//==================================================================================================
//								RJM Maszyny sp. z o.o.
//									13.05.2022
//	Obsługa silonwika podstawa z kontrolą czasów oraz kontrolą czujników
//	Realizacja wysuwania i chowania tłoczyska dla jednej cewki zwrócenie pozycji skrajnych
// 	v1.0	|| TC v 3.1.4024.22		|| - pierwsza wersja
//==================================================================================================
FUNCTION_BLOCK FB_Silownik_Kontola EXTENDS FB_Silownik 
VAR_INPUT
	stParametry								: DUT_SilownikParametry;
END_VAR
VAR_OUTPUT
END_VAR
VAR
	tonCzasNaPrace							: TON;
	tonCzasNaPowrot							: TON;
	fbKontrolaCzujnik0_F					: F_TRIG;
	fbKontrolaCzujnikMax_F					: F_TRIG;
	fbKontrolaCzujnik0_R					: R_TRIG;
	fbKontrolaCzujnikMax_R					: R_TRIG;
	fbLBKomunikacja							: FB_Silownik_Kontrola_Komunikacja;
END_VAR

METHOD Praca : BOOL
VAR_INPUT
END_VAR
SUPER^.Praca ();
//Czasy sprawdzające czas wysunięcia lub chowania tłoczyska
	tonCzasNaPrace (IN := bPrzesuwanieWStroneKonca, PT := REAL_TO_TIME (stParametry.rCzasNaPrace));
	tonCzasNaPowrot (In := bPrzesuwanieWStronePoczatku, PT := REAL_TO_TIME (stParametry.rCzasNaPowrot));
//kontrola wysuwania
	IF (tonCzasNaPrace.Q) THEN
		fbLBKomunikacja.UstawStan (iId := 1, bStan := TRUE);
	ELSIF (fbCzujnikPozycjaMax.CzyZadzialany AND NOT bPrzesuwanieWStroneKonca) THEN
		fbLBKomunikacja.UstawStan (iId := 1, bStan := FALSE);
	END_IF
//kontrola powrotu
	IF (tonCzasNaPowrot.Q) THEN
		fbLBKomunikacja.UstawStan (iId := 2, bStan := TRUE);
	ELSIF (fbCzujnikPozycja0.CzyZadzialany AND NOT bPrzesuwanieWStronePoczatku) THEN
		fbLBKomunikacja.UstawStan (iId := 2, bStan := FALSE);
	END_IF
//kontrola utraty pozycji 0
	fbKontrolaCzujnik0_F (CLK := fbCzujnikPozycja0.CzyZadzialany);
	IF (fbKontrolaCzujnik0_F.Q AND NOT bPrzesuwanieWStroneKonca) THEN
		fbLBKomunikacja.UstawStan (iId := 3, bStan := TRUE);
	ELSIF (fbCzujnikPozycja0.CzyZadzialany) THEN
		fbLBKomunikacja.UstawStan (iId := 3, bStan := FALSE);
	END_IF
//kontrola utraty pozycji MAX
	fbKontrolaCzujnikMax_F (CLK := fbCzujnikPozycjaMax.CzyZadzialany);
	IF (fbKontrolaCzujnikMax_F.Q AND NOT bPrzesuwanieWStronePoczatku) THEN
		fbLBKomunikacja.UstawStan (iId := 4, bStan := TRUE);
	ELSIF (fbCzujnikPozycjaMax.CzyZadzialany) THEN
		fbLBKomunikacja.UstawStan (iId := 4, bStan := FALSE);
	END_IF	
//Bladustawienia czujnikow - zadziałane dwa czujniki
	IF (fbCzujnikPozycja0.CzyZadzialany AND fbCzujnikPozycjaMax.CzyZadzialany) THEN
		fbLBKomunikacja.UstawStan (iId := 5, bStan := TRUE);
	ELSE
		fbLBKomunikacja.UstawStan (iId := 5, bStan := FALSE);
	END_IF
//Blad zamiany czujnikow	
	fbKontrolaCzujnik0_R (CLK := fbCzujnikPozycja0.CzyZadzialany);
	fbKontrolaCzujnikMax_R (CLK := fbCzujnikPozycjaMax.CzyZadzialany);
	IF ((fbKontrolaCzujnik0_R.Q AND bPrzesuwanieWStroneKonca) OR
		(fbKontrolaCzujnikMax_R.Q AND bPrzesuwanieWStronePoczatku)) THEN
		fbLBKomunikacja.UstawStan (iId := 6, bStan := FALSE);
	END_IF
	IF ((NaPoczatku AND NOT bPrzesuwanieWStroneKonca) OR 
		(NaKoncu and not bPrzesuwanieWStronePoczatku) ) THEN
		fbLBKomunikacja.UstawStan (iId := 6, bStan := FALSE);
	END_IF
END_METHOD

END_FUNCTION_BLOCK

(* stored: Version 1.1.0.1, ProductVersion 3.1.4024.11
   POU FB_Silownik_Kontola: Id {676285f5-d65d-4332-a0d9-89ca6ebe6eeb}, SpecialFunc None
   Method Praca: Id {5c9857db-7c66-48f3-9aab-6ac7209ef8b0} *)
